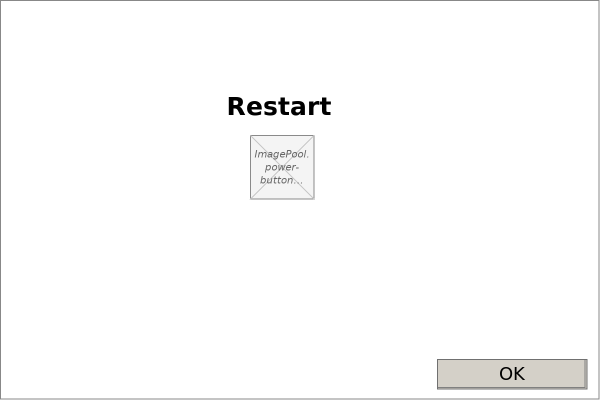
VISUALIZATION Dialog_Settings  // 600x400
    Button (437,359 150x30), "OK"
        OnMouseClick: CloseDialog Dialog=Dialog_Settings, Result=OK, NumpadKeypadSet=True
    Image (250,135 64x64), image: ImagePool.power-button-svgrepo-com
        OnMouseClick: toggle HMI.TC_Restart.RESTART
    Label (204,91 150x30), "Restart"
END_VISUALIZATION

(* stored: Version 1.1.0.1, ProductVersion 3.1.4024.3
   Visu Dialog_Settings: Id {163a6124-8c76-4037-b267-6a7ea0d6b5c4} *)
